// SIMATIC S7-200 project (STEP 7-Micro/WIN), CPU 221 REL 01.10

SYMBOL_TABLE USER1
CD_10S           I0.0
CD_20S           I0.1
CD_30S           I0.2
OFF              I0.3
DEN              Q0.0
END_SYMBOL_TABLE

ORGANIZATION_BLOCK MAIN:OB1
TITLE=
BEGIN
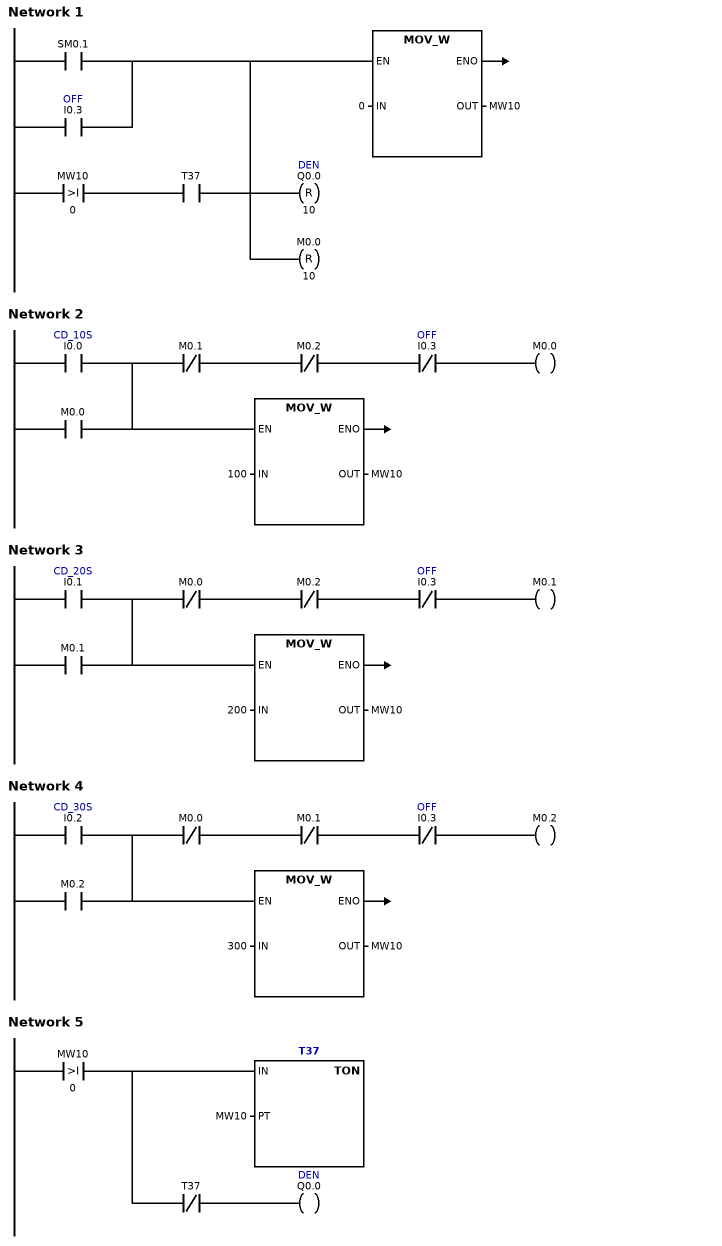
Network 1
LD     SM0.1
O      OFF:I0.3
LDW>   MW10, 0
A      T37
OLD
MOVW   0, MW10
R      DEN:Q0.0, 10
R      M0.0, 10
Network 2
LD     CD_10S:I0.0
O      M0.0
LPS
AN     M0.1
AN     M0.2
AN     OFF:I0.3
=      M0.0
LPP
MOVW   100, MW10
Network 3
LD     CD_20S:I0.1
O      M0.1
LPS
AN     M0.0
AN     M0.2
AN     OFF:I0.3
=      M0.1
LPP
MOVW   200, MW10
Network 4
LD     CD_30S:I0.2
O      M0.2
LPS
AN     M0.0
AN     M0.1
AN     OFF:I0.3
=      M0.2
LPP
MOVW   300, MW10
Network 5
LDW>   MW10, 0
TON    T37, MW10
AN     T37
=      DEN:Q0.0
END_ORGANIZATION_BLOCK
